% RSLogix 500 project Hands On 01.RSS, saved by version 10.00.00.00 %
PROJECT "UNTITLED"    % processor: Bul.1763 MicroLogix 1100 Series B %

PROGRAM FILES
  LAD 2   5 rungs

DATA FILES
  O0 OUTPUT  4 elements
  I1 INPUT  6 elements
  S2 STATUS  66 elements
  B3 BINARY  1 elements
  T4 TIMER  1 elements
  C5 COUNTER  1 elements
  R6 CONTROL  1 elements
  N7 INTEGER  1 elements
  F8 FLOAT  1 elements

LADDER 2
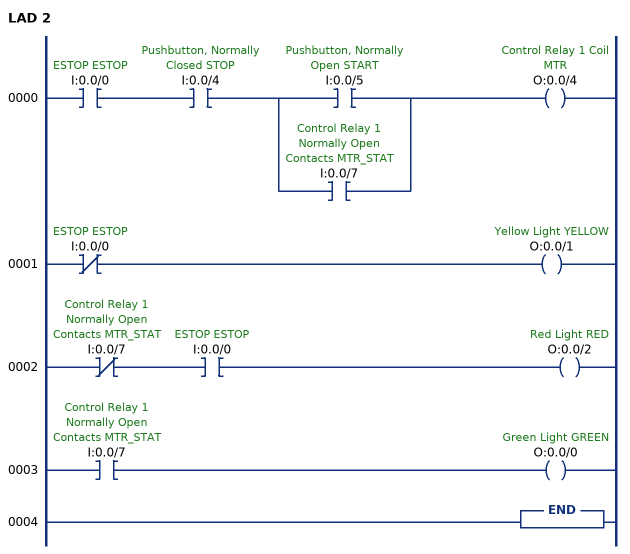
% Rung: 0 %
SOR XIC I:0.0/0 XIC I:0.0/4 BST XIC I:0.0/5 NXB XIC I:0.0/7 BND OTE O:0.0/4 EOR
%   I:0.0/0  ESTOP  "ESTOP" %
%   I:0.0/4  STOP  "Pushbutton, Normally Closed" %
%   I:0.0/5  START  "Pushbutton, Normally Open" %
%   I:0.0/7  MTR_STAT  "Control Relay 1 Normally Open Contacts" %
%   O:0.0/4  MTR  "Control Relay 1 Coil" %
% Rung: 1 %
SOR XIO I:0.0/0 OTE O:0.0/1 EOR
%   I:0.0/0  ESTOP  "ESTOP" %
%   O:0.0/1  YELLOW  "Yellow Light" %
% Rung: 2 %
SOR XIO I:0.0/7 XIC I:0.0/0 OTE O:0.0/2 EOR
%   I:0.0/7  MTR_STAT  "Control Relay 1 Normally Open Contacts" %
%   I:0.0/0  ESTOP  "ESTOP" %
%   O:0.0/2  RED  "Red Light" %
% Rung: 3 %
SOR XIC I:0.0/7 OTE O:0.0/0 EOR
%   I:0.0/7  MTR_STAT  "Control Relay 1 Normally Open Contacts" %
%   O:0.0/0  GREEN  "Green Light" %
% Rung: 4 %
SOR END EOR
